ABB RobotStudio station: comportamiento_real_2.rspag

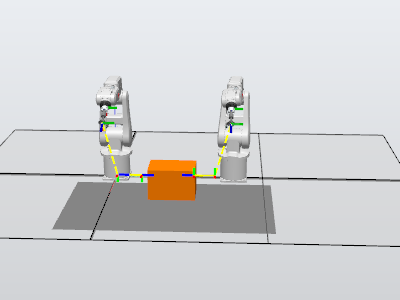
--- station ---
Station comportamiento1 (saved by RobotStudio 25.1.11133.0)
Controller IRB120_3_58_1, task T_ROB1: task frame (RAPID world) sits at (0, 800, 0) mm in the station
Controller IRB120_3_58
  mechanical unit ROB_1: IRB120_3_58__01, 6 joints, base frame (0, 0, 0) mm
Controller IRB120_3_58_1
  mechanical unit ROB_1: IRB120_3_58__02, 6 joints, base frame (0, 0, 0) mm
Layout (positions relative to the parent item):
  - IRB120_3_58__01 [mechanism, from %ABB.RobotStudio.Models.IRB120%\IRB120_3_58_G_01.rslib] at (0, 0, 0) mm; joint values [0, 0, 0, 0, 0.5236, 0] (rad or m)
  - IRB120_3_58__02 [mechanism, from %ABB.RobotStudio.Models.IRB120%\IRB120_3_58_G_01.rslib] at (0, 800, 0) mm; joint values [-0.0918, -0.3344, 0.3612, 0.165, 0.5044, -0.1907] (rad or m)
  - SC_VentosaD50_6 [smart component, from Components\SC_VentosaD50.rslib] at (364.35, 0, 594) mm, rotated rx 180 ry 60 rz 180 deg
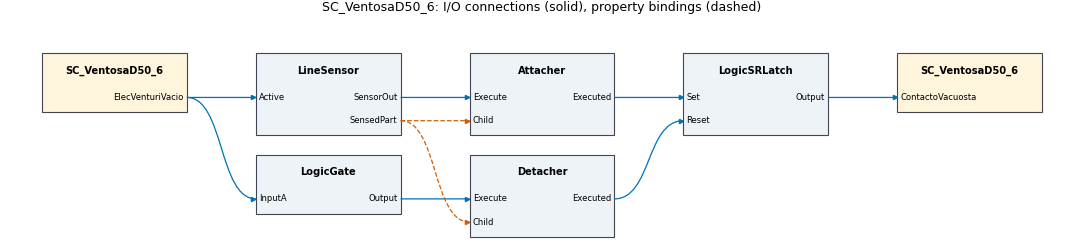
      connections:
        SC_VentosaD50_6.ElecVenturiVacio -> LineSensor.Active
        LineSensor.SensorOut -> Attacher.Execute
        Attacher.Executed -> LogicSRLatch.Set
        LogicSRLatch.Output -> SC_VentosaD50_6.ContactoVacuostato
        SC_VentosaD50_6.ElecVenturiVacio -> LogicGate.InputA
        LogicGate.Output -> Detacher.Execute
        Detacher.Executed -> LogicSRLatch.Reset
        LineSensor.SensedPart => Attacher.Child
        LineSensor.SensedPart => Detacher.Child
    - ToolVentosaD50 [mechanism, from Components\SC_VentosaD50.rslib] at (0, 0, 0) mm
    - Attacher [smart component, from Components\Attacher.rslib]
        properties: Parent=ToolVentosaD50; Flange=0; Child=Pieza_6; Mount=false; Offset=[0 0 0]; Orientation=[0 0 0]
    - Detacher [smart component, from Components\Detacher.rslib]
        properties: Child=Pieza_6; KeepPosition=true
    - LineSensor [smart component, from Components\LineSensor.rslib] at (0, 0, 126) mm
        properties: Start=[0 0 0]; End=[0 0 0.015]; Radius=0.001; SensedPart=Pieza_6; SensedPoint=[0.310468994140625 0.257791259765625 0.100099983215332]; Length=0.015; Tag=(none); SenseMultiple=false
      - _sensorPart_ [part], size 2 x 2 x 15 mm
    - LogicGate [smart component, from Components\LogicGate.rslib]
        properties: Operator=NOT; Delay=0
    - LogicSRLatch [smart component, from Components\LogicSRLatch.rslib]
  - SC_VentosaD50_7 [smart component, from Components\SC_VentosaD50.rslib] at (276.59, 780.28, 570.93) mm, rotated rx -180 ry 60 rz -180 deg
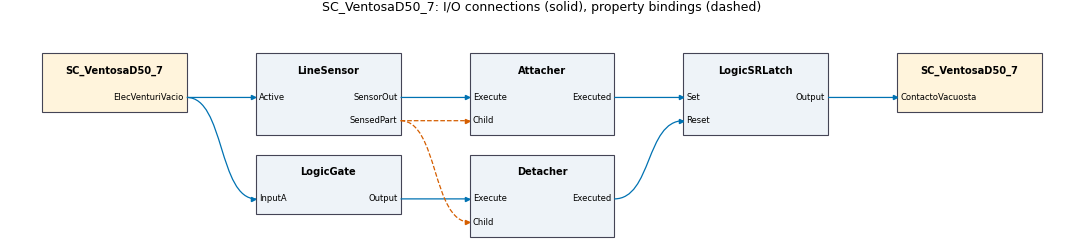
      connections:
        SC_VentosaD50_7.ElecVenturiVacio -> LineSensor.Active
        LineSensor.SensorOut -> Attacher.Execute
        Attacher.Executed -> LogicSRLatch.Set
        LogicSRLatch.Output -> SC_VentosaD50_7.ContactoVacuostato
        SC_VentosaD50_7.ElecVenturiVacio -> LogicGate.InputA
        LogicGate.Output -> Detacher.Execute
        Detacher.Executed -> LogicSRLatch.Reset
        LineSensor.SensedPart => Attacher.Child
        LineSensor.SensedPart => Detacher.Child
    - ToolVentosaD50 [mechanism, from Components\SC_VentosaD50.rslib] at (0, 0, 0) mm
    - Attacher [smart component, from Components\Attacher.rslib]
        properties: Parent=ToolVentosaD50; Flange=0; Child=(none); Mount=false; Offset=[0 0 0]; Orientation=[0 0 0]
    - Detacher [smart component, from Components\Detacher.rslib]
        properties: Child=(none); KeepPosition=true
    - LineSensor [smart component, from Components\LineSensor.rslib] at (0, 0, 126) mm
        properties: Start=[0 0 0]; End=[0 0 0.015]; Radius=0.001; SensedPart=(none); SensedPoint=[0 0 0]; Length=0.015; Tag=(none); SenseMultiple=false
      - _sensorPart_ [part], size 2 x 2 x 15 mm
    - LogicGate [smart component, from Components\LogicGate.rslib]
        properties: Operator=NOT; Delay=0
    - LogicSRLatch [smart component, from Components\LogicSRLatch.rslib]
  - LogicGate [smart component, from Components\LogicGate.rslib]
      properties: Operator=AND; Delay=0
  - Pieza_2 [part], size 750 x 1300 x 0.1 mm
  - Pieza_6 [part] at (88.62, -142.22, -0.16) mm, rotated rx -0.05 ry -0.19 rz 0.1 deg, size 200 x 300 x 200 mm
Attachment: SC_VentosaD50_6 is attached to IRB120_3_58__01 / Link6
Attachment: SC_VentosaD50_7 is attached to IRB120_3_58__02 / Link6
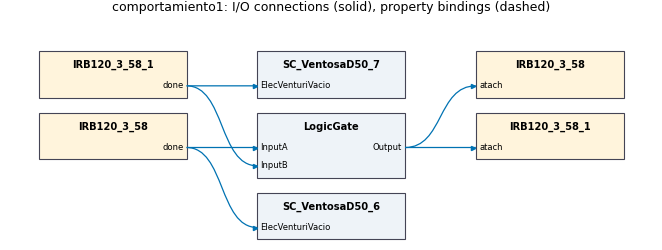
Station logic (signal -> signal, property => property):
  IRB120_3_58_1.done -> SC_VentosaD50_7.ElecVenturiVacio
  IRB120_3_58.done -> SC_VentosaD50_6.ElecVenturiVacio
  IRB120_3_58.done -> LogicGate.InputA
  IRB120_3_58_1.done -> LogicGate.InputB
  LogicGate.Output -> IRB120_3_58.atach
  LogicGate.Output -> IRB120_3_58_1.atach

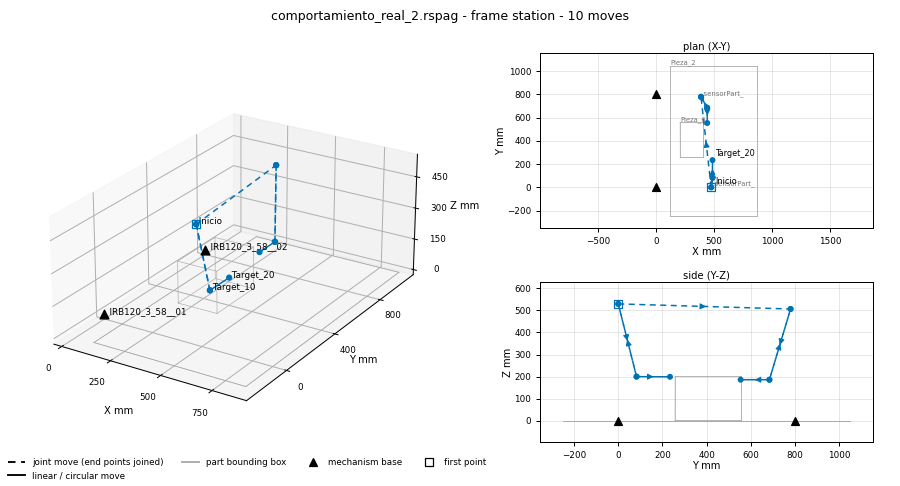
[picture p0: tool path of comportamiento_real_2.rspag in frame station, 10 of 14 moves have a stored position in this frame; points joined in program order, loops and branches not executed]
--- Controller Data/IRB120_3_58/RAPID/TASK1/PROGMOD/CalibData.mod ---
MODULE CalibData
    PERS tooldata TCP_ToolVentosaD50:=[TRUE,[[0,0,129.5],[1,0,0,0]],[1,[0,0,1],[1,0,0,0],0,0,0]];
ENDMODULE

--- Controller Data/IRB120_3_58/RAPID/TASK1/PROGMOD/Module1.mod ---
MODULE Module1
        CONST robtarget Inicio:=[[476.504118863,0,529.25],[0.5,0,0.866025404,0],[0,0,0,0],[9E+09,9E+09,9E+09,9E+09,9E+09,9E+09]];
    CONST robtarget Target_10:=[[488.12,82.71,199.94],[0.707106781,-0.707106781,0,0],[-1,0,1,0],[9E+09,9E+09,9E+09,9E+09,9E+09,9E+09]];
    CONST robtarget Target_20:=[[488.05,234.27,199.06],[0.707106781,-0.707106781,0,0],[0,1,0,0],[9E+09,9E+09,9E+09,9E+09,9E+09,9E+09]];

    VAR socketdev server1;
    VAR socketdev clientSocket;
    VAR bool Z_1;
    VAR string data1;
    VAR num cambioStrZ;
    VAR string ZValorString;

    VAR num PZ:=0;

    PROC main()

        SocketCreate server1;
        SocketBind server1, "127.0.0.1", 8000;
        SocketListen server1;
        SocketAccept server1, clientSocket, \Time:=WAIT_MAX;
        SocketSend clientSocket \str:= "Conexion ABB 1";

        Path_10;
    ENDPROC

    PROC Path_10()
        MoveJ Inicio,v50,fine,TCP_ToolVentosaD50\WObj:=wobj0;
        SocketSend clientSocket \str:= "1";
        SocketReceive clientSocket \str:= data1;
        MoveJ Target_10,v50,fine,TCP_ToolVentosaD50\WObj:=wobj0;
        SocketSend clientSocket \str:= "1";
        SocketReceive clientSocket \str:= data1;
        MoveL Target_20,v50,fine,TCP_ToolVentosaD50\WObj:=wobj0;
        SocketSend clientSocket \str:= "1";

        FOR i FROM 1 TO 7 DO
            SocketReceive clientSocket \str:= data1;
            PZ := PZ+50;
            MoveL Offs(Target_20,0,0,PZ),v50,fine,TCP_ToolVentosaD50\WObj:=wobj0;
            SocketSend clientSocket \str:= "1";
        ENDFOR
        !PZ :=0;
        FOR i FROM 1 TO 7 DO
            SocketReceive clientSocket \str:= data1;
            PZ := PZ-50;
            MoveL Offs(Target_20,0,0,PZ),v50,fine,TCP_ToolVentosaD50\WObj:=wobj0;
            SocketSend clientSocket \str:= "1";
        ENDFOR

        SocketReceive clientSocket \str:= data1;
        MoveL Target_10,v50,fine,TCP_ToolVentosaD50\WObj:=wobj0;
        SocketSend clientSocket \str:= "1";
        SocketReceive clientSocket \str:= data1;
        MoveJ Inicio,v50,fine,TCP_ToolVentosaD50\WObj:=wobj0;
        SocketSend clientSocket \str:= "1";
    ENDPROC
ENDMODULE

--- Controller Data/IRB120_3_58_1/RAPID/TASK1/PROGMOD/Module1.mod ---
MODULE Module1
        CONST robtarget Inicio:=[[388.74,-19.72,506.18],[0.5,0,0.866025404,0],[0,0,0,0],[9E+09,9E+09,9E+09,9E+09,9E+09,9E+09]];
    CONST robtarget Target_10:=[[442.77,-115.57,185.9],[0.707106781,0.707106781,0,0],[0,-1,-2,0],[9E+09,9E+09,9E+09,9E+09,9E+09,9E+09]];
    CONST robtarget Target_20:=[[442.78,-245.8,185.89],[0.707106781,0.707106781,0,0],[-1,-2,-1,0],[9E+09,9E+09,9E+09,9E+09,9E+09,9E+09]];

    VAR socketdev server2;
    VAR socketdev clientSocket2;
    VAR string data2;
    VAR num PZ:=0;

    PROC main()

        SocketCreate server2;
        SocketBind server2, "127.0.0.2", 8000;
        SocketListen server2;
        SocketAccept server2, clientSocket2, \Time:=WAIT_MAX;
        SocketSend clientSocket2 \str:= "Conexion ABB 2";

        Path_10;
    ENDPROC

    PROC Path_10()
        MoveJ Inicio,v50,fine,TCP_ToolVentosaD50\WObj:=wobj0;
        SocketSend clientSocket2 \str:= "2";
        SocketReceive clientSocket2 \str:= data2;
        MoveJ Target_10,v50,fine,TCP_ToolVentosaD50\WObj:=wobj0;
        SocketSend clientSocket2 \str:= "2";
        SocketReceive clientSocket2 \str:= data2;
        MoveL Target_20,v50,fine,TCP_ToolVentosaD50\WObj:=wobj0;
        SocketSend clientSocket2 \str:= "2";

        FOR i FROM 1 TO 7 DO
            SocketReceive clientSocket2 \str:= data2;
            PZ := PZ+50;
            MoveL Offs(Target_20,0,0,PZ),v50,fine,TCP_ToolVentosaD50\WObj:=wobj0;
            SocketSend clientSocket2 \str:= "2";
        ENDFOR
        !PZ :=0;
        FOR i FROM 1 TO 7 DO
            SocketReceive clientSocket2 \str:= data2;
            PZ := PZ-50;
            MoveL Offs(Target_20,0,0,PZ),v50,fine,TCP_ToolVentosaD50\WObj:=wobj0;
            SocketSend clientSocket2 \str:= "2";
        ENDFOR

        SocketReceive clientSocket2 \str:= data2;
        MoveL Target_10,v50,fine,TCP_ToolVentosaD50\WObj:=wobj0;
        SocketSend clientSocket2 \str:= "2";
        SocketReceive clientSocket2 \str:= data2;
        MoveJ Inicio,v50,fine,TCP_ToolVentosaD50\WObj:=wobj0;
        SocketSend clientSocket2 \str:= "2";
    ENDPROC
ENDMODULE

--- Controller Data/IRB120_3_58/SYSPAR/EIO.cfg ---
EIO:CFG_1.0:6:1::
#
EIO_SIGNAL:

      -Name "done" -SignalType "DO"

      -Name "atach" -SignalType "DI"
